FUNCTION_BLOCK TN_SC_AREA_SAVE
VAR
	in_Offset_1 : INT;
	in_Offset_2 : INT;
	in_Y : INT;
	in_X : INT;
END_VAR
VAR_INPUT
	Iin_Y1 : INT;
	Iin_X1 : INT;
	Iin_Y2 : INT;
	Iin_X2 : INT;
END_VAR
VAR_IN_OUT
	Xus_TN_SCREEN : us_TN_SCREEN;
END_VAR

(*
version 1.0		10. mai 2010
programmer		ks
tested by		ks

TN_SC_AREA_SAVE sichert den angegebenen Bildschirmbereich in einem Buffer
*)

IF TN_SC_XY2_ERROR(Iin_X1,Iin_Y1,Iin_X2,Iin_Y2) THEN RETURN; END_IF;

(* Parameter ablegen *)
Xus_TN_SCREEN.bya_BACKUP[0] := BYTE#1;
Xus_TN_SCREEN.bya_BACKUP[1] := INT_TO_BYTE(Iin_X1);
Xus_TN_SCREEN.bya_BACKUP[2] := INT_TO_BYTE(Iin_Y1); 
Xus_TN_SCREEN.bya_BACKUP[3] := INT_TO_BYTE(Iin_X2);
Xus_TN_SCREEN.bya_BACKUP[4] := INT_TO_BYTE(Iin_Y2);

in_Offset_2 := 5;
(* CHAR und COLOR in BUFFER sichern *)
FOR in_Y := Iin_Y1 TO Iin_Y2 DO

	in_Offset_1 := (in_Y * 80) + Iin_X1;
	FOR in_X := Iin_X1 TO Iin_X2 DO
		Xus_TN_SCREEN.bya_BACKUP[in_Offset_2] := Xus_TN_SCREEN.bya_CHAR[in_Offset_1];
		in_Offset_2 := in_Offset_2 + INT#01;
		Xus_TN_SCREEN.bya_BACKUP[in_Offset_2] := Xus_TN_SCREEN.bya_COLOR[in_Offset_1];
		in_Offset_2 := in_Offset_2 + INT#01;
		in_Offset_1 := in_Offset_1 + INT#01;
	END_FOR;
END_FOR;

(* revision history
ks	10. mai. 2010	rev 1.0
	original version
*)

END_FUNCTION_BLOCK

(* stored: Version 1.1.0.1, ProductVersion 3.1.4024.0
   POU TN_SC_AREA_SAVE: Id {2bc40e97-3444-4d05-b071-ce96da9a895d}, SpecialFunc None *)
